# EPICS substitutions: sairemai4s-loc/sairemai4sApp/Db/sairemai4s.substitutions
file sairemai4s.template
{
    {
        secsub    = ISrc-010,
        disdevidx = ISS-ATU,
        write     = sai4s-modbus-write-word,
        read      = sai4s-modbus-read-word
    }
}
